PROGRAM P_Demo_FB_DMXGetSupportedParameters
VAR
    fbGetSupported    : FB_DMXGetSupportedParameters; // 读支持的 PID 列表
    stDmxCmdBuffer    : ST_DMXCommandBuffer;          // 与通讯 FB 共用
    wTargetManufId    : WORD := 16#4241;              // 目标灯具厂商 ID
    dwTargetDeviceId  : DWORD := 16#12131415;         // 目标灯具设备 ID
    byTargetPort      : BYTE := 0;                    // 根设备通道 0
    bDoRead           : BOOL := FALSE;                // 在线给一次上升沿触发
    bBusy             : BOOL;
    bError            : BOOL;
    udiErrId          : UDINT;
    arrSupportedPids  : ARRAY [0..114] OF E_DMXParameterId;  // 支持的 PID 列表
END_VAR

// ============================================================
// Tc2_DMX.FB_DMXGetSupportedParameters 演示程序
// ============================================================
// 场景：通用上位机适配设备：先读支持的 PID 列表，据此动态启用/隐藏功能按钮。
// 价值：把设备能力清单从设备直接读出，实现按能力裁剪的自适应界面与控制逻辑，避免盲发命令报错。
// 验证：给 bDoRead 一次上升沿 -> bBusy 短暂 TRUE -> 回 FALSE 后 arrSupportedPids 列出设备支持的可选 PID（数组前若干元素有效）。
// 验证步骤：
//   1. 右键 PLC 项目下 POUs 文件夹 → Add → Existing Item → 选本 .TcPOU 文件
//   2. 引用 Tc2_DMX；同项目里放一个 FB_EL6851CommunicationEx 实例并共用 stDmxCmdBuffer（非 CycleMode）
//   3. 编译 → 登录 → 运行；按上方『验证』行在线给上升沿观察
// ============================================================

fbGetSupported(
    bStart                     := bDoRead,
    wDestinationManufacturerId := wTargetManufId,
    dwDestinationDeviceId      := dwTargetDeviceId,
    byPortId                   := byTargetPort,
    dwOptions                  := 0,
    stCommandBuffer            := stDmxCmdBuffer,
    bBusy                      => bBusy,
    bError                     => bError,
    udiErrorId                 => udiErrId,
    arrParameters              => arrSupportedPids
);

END_PROGRAM

(* stored: Version 1.1.0.1, ProductVersion 3.1.4024.5
   POU P_Demo_FB_DMXGetSupportedParameters: Id {c2851e7d-2eaf-55c0-b73a-2f7206d91632}, SpecialFunc None *)
